FUNCTION Camera_Set_Input_Layout : UINT
VAR_INPUT
	Layout : Buffer_Layout;
END_VAR
VAR_IN_OUT
	Camera : Cognex_Camera;
END_VAR

Camera.Input_Buffer_Layout := Layout;

END_FUNCTION

(* stored: Version 1.1.0.1, ProductVersion 3.1.4024.10
   POU Camera_Set_Input_Layout: Id {85060792-d177-4be9-9036-bbab4b2e6963}, SpecialFunc None *)
